{attribute 'GeneratedUsingTerminal: EL4021-0000-0016'}
{attribute addProperty BoxType "EL4021-0000-0016"}
{attribute addProperty Description "EL4021 1Ch. Ana. Output 4-20mA, 12bit"}
{attribute addProperty Physics "KK"}
{attribute addProperty Id "AO_OutputsAT %Q*AO_Output_Channel_BA7EBB7C2WcStateAT %I*WcState_0B2B16F91InfoDataAT %I*InfoData_32EB74EA10"}
{attribute addProperty CRC "3024842059"}
{attribute addProperty Size "13"}
TYPE EL4021_B44B6D4B EXTENDS EtcSlaveTerminalBase_947E5A46 :
STRUCT
	{attribute addProperty Name "AO_Outputs"}
	AO_Outputs : AO_Output_Channel_BA7EBB7C;
	{attribute addProperty Name "WcState"}
	WcState : WcState_0B2B16F9;
	{attribute addProperty Name "InfoData"}
	InfoData : InfoData_32EB74EA;
END_STRUCT
END_TYPE

(* stored: Version 1.2.0.0, ProductVersion 3.1.4024.9
   DUT EL4021_B44B6D4B: Id {bad5ff42-9412-43d9-a36f-725d4b9c713b} *)
